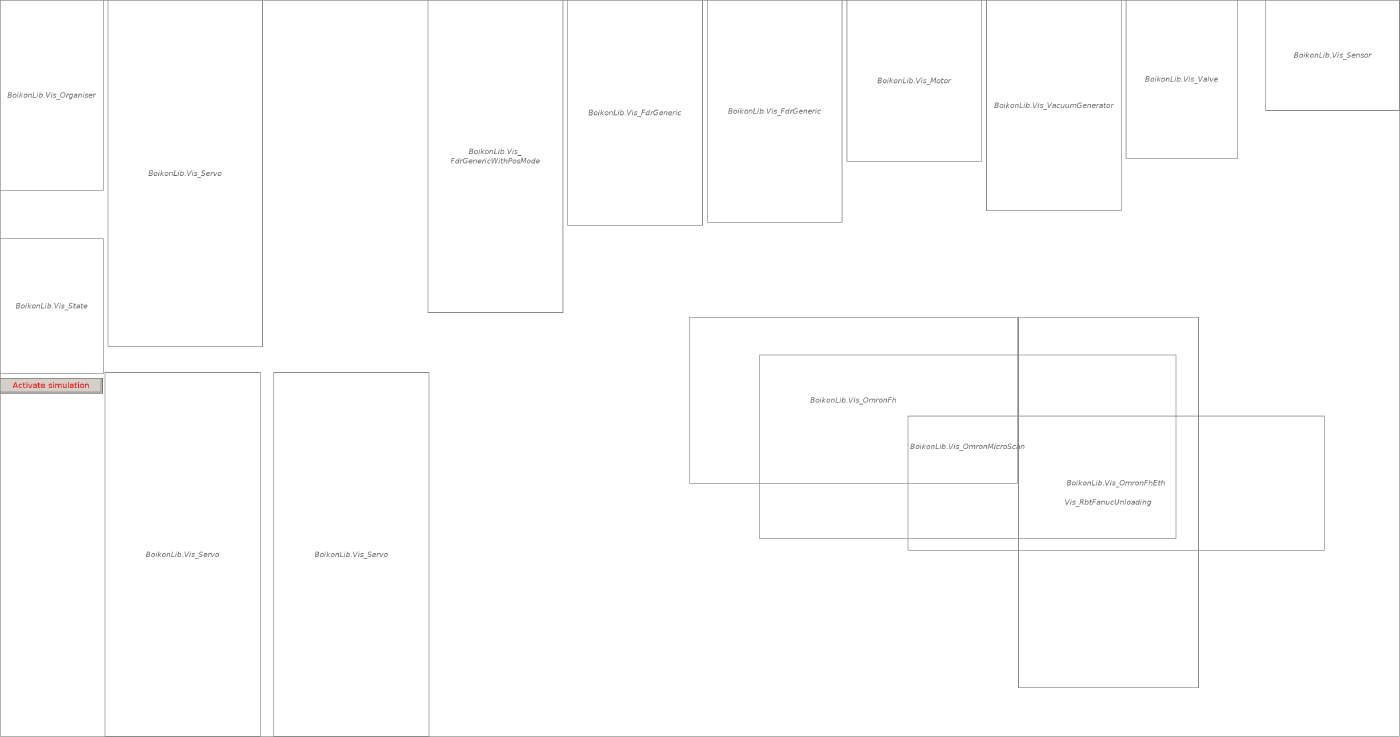
VISUALIZATION VisScmTemplate  // 1925x1014
    Frame (148,0 213x477)
        shows BoikonLib.Vis_Servo(I_UnitName := 'Xaxis', IO_cntrl_Servo := MAIN.ExampleMachinePart.Srv_Xaxis)
    Button (0,520 141x21), "Activate simulation"
        toggle Glbl.Sim_MyMachinePart
    Frame (1044,488 573x253)
        shows BoikonLib.Vis_OmronMicroScan(I_UnitName := 'Omron Smart Cam', IO_cntrl := MAIN.ExampleMachinePart.Cam_OmronSmartCam)
    Frame (948,436 451x229)
        shows BoikonLib.Vis_OmronFh(I_UnitName := 'OmronFh', IO_cntrl := MAIN.ExampleMachinePart.Cam_OmronFh)
    Frame (1740,0 185x152)
        shows BoikonLib.Vis_Sensor(I_UnitName := 'Example sensor', IO_cntrl := MAIN.ExampleMachinePart.PC_ProductInfeed)
    Frame (1548,0 154x218)
        shows BoikonLib.Vis_Valve(I_UnitName := 'TempValve', IO_cntrl := MAIN.ExampleMachinePart.Cyl_Example)
    Frame (1356,0 186x290)
        shows BoikonLib.Vis_VacuumGenerator(I_UnitName := 'VacuumGenerator', IO := MAIN.ExampleMachinePart.Vcg_Suckers)
    Frame (1248,572 573x185)
        shows BoikonLib.Vis_OmronFhEth(I_UnitName := 'OmronEth', IO_cntrl := MAIN.ExampleMachinePart.Cam_OmronFhEth)
    Frame (972,0 186x306)
        shows BoikonLib.Vis_FdrGeneric(I_UnitName := 'Lenze', IO_Cntrl := MAIN.ExampleMachinePart.Fdr_LzExample)
    Frame (780,0 186x310)
        shows BoikonLib.Vis_FdrGeneric(I_UnitName := 'ControlTech', IO_Cntrl := MAIN.ExampleMachinePart.Fdr_CtExample)
    Frame (1164,0 186x222)
        shows BoikonLib.Vis_Motor(I_UnitName := 'Example', IO_cntrl := MAIN.ExampleMachinePart.Mtr_Example)
    Frame (0,0 142x262)
        shows BoikonLib.Vis_Organiser(I_UnitName := 'Organiser'', IO_cntrl_Organiser := MAIN.Organiser)
    Frame (588,0 186x430)
        shows BoikonLib.Vis_FdrGenericWithPosMode(I_UnitName := 'Interrol', IO_Cntrl := MAIN.ExampleMachinePart.Srv_Interrol)
    Frame (0,328 142x186)
        shows BoikonLib.Vis_State(I_UnitName := 'SCM state', IO_Step := MAIN.ExampleMachinePart.State)
    Frame (1400,436 248x510)
        shows Vis_RbtFanucUnloading(I_UnitName := 'Unloading', IO_cntrl := MAIN.ExampleMachinePart.Rbt_Unloading)
    Frame (144,512 214x502)
        shows BoikonLib.Vis_Servo(I_UnitName := 'Yaxis', IO_cntrl_Servo := MAIN.ExampleMachinePart.Srv_Yaxis)
    Frame (376,512 214x502)
        shows BoikonLib.Vis_Servo(I_UnitName := 'Zaxis', IO_cntrl_Servo := MAIN.ExampleMachinePart.Srv_Zaxis)
END_VISUALIZATION

(* stored: Version 1.1.0.1
   Visu VisScmTemplate: Id {e955b262-be3e-40c0-8bd4-c1c40ccdad65} *)
